# EPICS autosave request: iocBoot/gmca_23o_ioc1/dbSave/bluiceClient.req
$(P)mode
$(P)pid
$(P)host
$(P)user
$(P)state
